IP02: A     #t_Safety_Pwr_On_GRP16;
      AN    #t_Suppress_Errors;
      AN    #t_Suppress_Errors_Isafe;
      AN    #s_Status.THO_Main_Pwr_GRP16;
      AN    #s_Status.No_Power_GRP16;
      AN    #s_Status.THO_Aux_Pwr_GRP16;
      A     #i_CFG_Motor_Prsnt_GRP16;
      =     #s_Motor_Grp.Motor_Group_16_in;
NETWORK
TITLE =JA: Safety Signal Handling
//Handle safety stop signals for every motor group
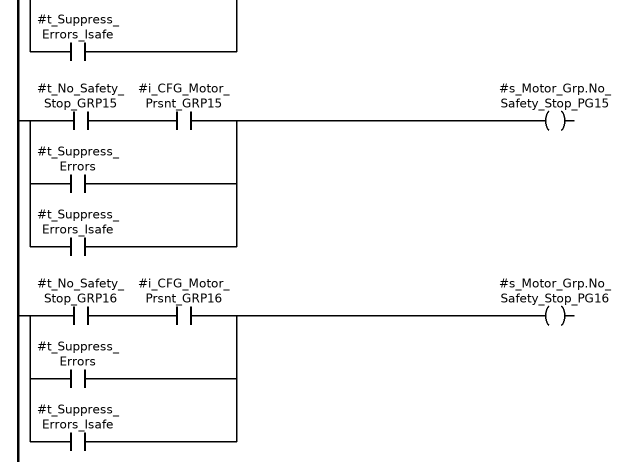
      NOP   0;
// No Safety stop MotorGroup 01
      A     #t_No_Safety_Stop_GRP01;
      A     #i_CFG_Motor_Prsnt_GRP01;
      O     #t_Suppress_Errors;
      O     #t_Suppress_Errors_Isafe;
      =     #s_Motor_Grp.No_Safety_Stop_PG01;

// No Safety stop MotorGroup 02
      A     #t_No_Safety_Stop_GRP02;
      A     #i_CFG_Motor_Prsnt_GRP02;
      O     #t_Suppress_Errors;
      O     #t_Suppress_Errors_Isafe;
      =     #s_Motor_Grp.No_Safety_Stop_PG02;

// No Safety stop MotorGroup 03
      A     #t_No_Safety_Stop_GRP03;
      A     #i_CFG_Motor_Prsnt_GRP03;
      O     #t_Suppress_Errors;
      O     #t_Suppress_Errors_Isafe;
      =     #s_Motor_Grp.No_Safety_Stop_PG03;

// No Safety stop MotorGroup 04
      A     #t_No_Safety_Stop_GRP04;
      A     #i_CFG_Motor_Prsnt_GRP04;
      O     #t_Suppress_Errors;
      O     #t_Suppress_Errors_Isafe;
      =     #s_Motor_Grp.No_Safety_Stop_PG04;

// No Safety stop MotorGroup 05
      A     #t_No_Safety_Stop_GRP05;
      A     #i_CFG_Motor_Prsnt_GRP05;
      O     #t_Suppress_Errors;
      O     #t_Suppress_Errors_Isafe;
      =     #s_Motor_Grp.No_Safety_Stop_PG05;

// No Safety stop MotorGroup 06
      A     #t_No_Safety_Stop_GRP06;
      A     #i_CFG_Motor_Prsnt_GRP06;
      O     #t_Suppress_Errors;
      O     #t_Suppress_Errors_Isafe;
      =     #s_Motor_Grp.No_Safety_Stop_PG06;

// No Safety stop MotorGroup 07
      A     #t_No_Safety_Stop_GRP07;
      A     #i_CFG_Motor_Prsnt_GRP07;
      O     #t_Suppress_Errors;
      O     #t_Suppress_Errors_Isafe;
      =     #s_Motor_Grp.No_Safety_Stop_PG07;

// No Safety stop MotorGroup 08
      A     #t_No_Safety_Stop_GRP08;
      A     #i_CFG_Motor_Prsnt_GRP08;
      O     #t_Suppress_Errors;
      O     #t_Suppress_Errors_Isafe;
      =     #s_Motor_Grp.No_Safety_Stop_PG08;

// No Safety stop MotorGroup 09
      A     #t_No_Safety_Stop_GRP09;
      A     #i_CFG_Motor_Prsnt_GRP09;
      O     #t_Suppress_Errors;
      O     #t_Suppress_Errors_Isafe;
      =     #s_Motor_Grp.No_Safety_Stop_PG09;

// No Safety stop MotorGroup 10
      A     #t_No_Safety_Stop_GRP10;
      A     #i_CFG_Motor_Prsnt_GRP10;
      O     #t_Suppress_Errors;
      O     #t_Suppress_Errors_Isafe;
      =     #s_Motor_Grp.No_Safety_Stop_PG10;

// No Safety stop MotorGroup 11
      A     #t_No_Safety_Stop_GRP11;
      A     #i_CFG_Motor_Prsnt_GRP11;
      O     #t_Suppress_Errors;
      O     #t_Suppress_Errors_Isafe;
      =     #s_Motor_Grp.No_Safety_Stop_PG11;

// No Safety stop MotorGroup 12
      A     #t_No_Safety_Stop_GRP12;
      A     #i_CFG_Motor_Prsnt_GRP12;
      O     #t_Suppress_Errors;
      O     #t_Suppress_Errors_Isafe;
      =     #s_Motor_Grp.No_Safety_Stop_PG12;

// No Safety stop MotorGroup 13
      A     #t_No_Safety_Stop_GRP13;
      A     #i_CFG_Motor_Prsnt_GRP13;
      O     #t_Suppress_Errors;
      O     #t_Suppress_Errors_Isafe;
      =     #s_Motor_Grp.No_Safety_Stop_PG13;

// No Safety stop MotorGroup 14
      A     #t_No_Safety_Stop_GRP14;
      A     #i_CFG_Motor_Prsnt_GRP14;
      O     #t_Suppress_Errors;
      O     #t_Suppress_Errors_Isafe;
      =     #s_Motor_Grp.No_Safety_Stop_PG14;

// No Safety stop MotorGroup 15
      A     #t_No_Safety_Stop_GRP15;
      A     #i_CFG_Motor_Prsnt_GRP15;
      O     #t_Suppress_Errors;
      O     #t_Suppress_Errors_Isafe;
      =     #s_Motor_Grp.No_Safety_Stop_PG15;

// No Safety stop MotorGroup 16
      A     #t_No_Safety_Stop_GRP16;
      A     #i_CFG_Motor_Prsnt_GRP16;
      O     #t_Suppress_Errors;
      O     #t_Suppress_Errors_Isafe;
      =     #s_Motor_Grp.No_Safety_Stop_PG16;

NETWORK
TITLE =KA: Copy motor group status to DB

      OPN   #i_DB_Motor_Slave;

      L     DBNO;
      T     #t_DB_NO;

      L     DBLG;
      T     #t_DB_Length;

// define t_ANY_data
      LAR1  P##t_ANY_DB_Motor_Slave; // input ANY POINTER

// Copy the the pointer type to the Temporary pointers
      L     W#16#1002; // ANY pointer type: 10 for S7, 02 for data type 'BYTE'
      T     LW [AR1,P#0.0]; // ANY pointer type

// Copy the repetition factor (= data lentgh) to the Temporary pointers
      L     #t_DB_Length; // Number of bytes to copy
      T     LW [AR1,P#2.0]; // ANY pointer repetition factor

// Copy the DB number to the Data temporary pointer
      L     #t_DB_NO; // ANY POINTER for data to write
      T     LW [AR1,P#4.0]; // ANY pointer DB number

// Copy the Area pointer to the Data Temporary pointer
      L     0;
      T     LD [AR1,P#6.0]; // ANY pointer Area pointer
      L     B#16#84; //Store 84H: DB Global data area in ANY
      T     LB [AR1,P#6.0];

      CALL "BLKMOV" (
           SRCBLK                   := #s_Motor_Grp,
           RET_VAL                  := #t_Ret_Val,
           DSTBLK                   := #t_ANY_DB_Motor_Slave);

NETWORK
TITLE =LA: Handle commands
//Set the controlled stop and direct stop output signals.
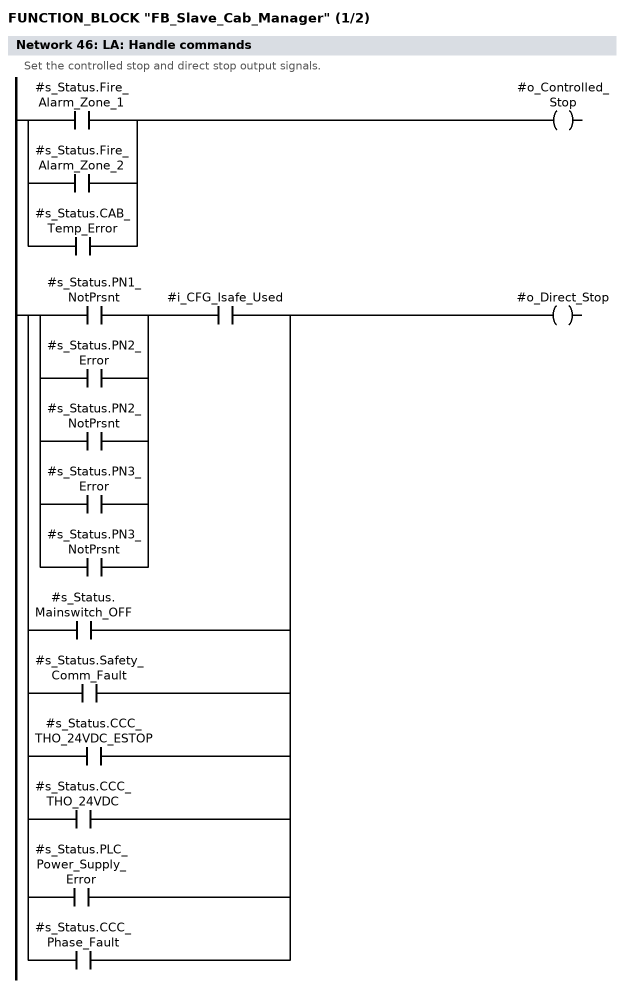
      O     #s_Status.Fire_Alarm_Zone_1;
      O     #s_Status.Fire_Alarm_Zone_2;
      O     #s_Status.CAB_Temp_Error;
      =     #o_Controlled_Stop;

      A(    ;
      O     #s_Status.PN1_NotPrsnt;
      O     #s_Status.PN2_Error;
      O     #s_Status.PN2_NotPrsnt;
      O     #s_Status.PN3_Error;
      O     #s_Status.PN3_NotPrsnt;
      )     ;
      A     #i_CFG_Isafe_Used;
      O     #s_Status.Mainswitch_OFF;
      O     #s_Status.Safety_Comm_Fault;
      O     #s_Status.CCC_THO_24VDC_ESTOP;
      O     #s_Status.CCC_THO_24VDC;
      O     #s_Status.PLC_Power_Supply_Error;
// Option to stop is Phase fault is detected.
      O     #s_Status.CCC_Phase_Fault;
      =     #o_Direct_Stop;
NETWORK
TITLE =MA: Write output signals
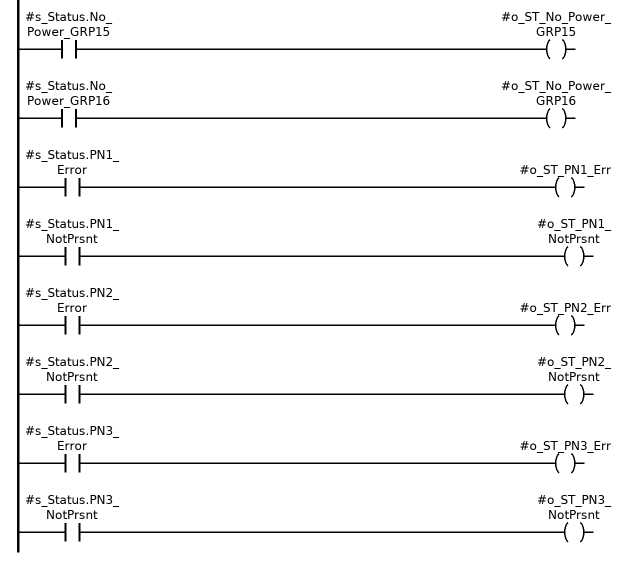

      A     #s_Status.Mainswitch_OFF;
      =     #o_ST_Mainswitch_OFF;

      A     #s_Status.Safety_Comm_Fault;
      =     #o_ST_Safety_Comm_Fault;

      A     #s_Status.CCC_THO_24VDC;
      =     #o_ST_CCC_THO_1_24VDC;

      A     #s_Status.PLC_Power_Supply_Error;
      =     #o_ST_CCC_THO_2_24VDC;

      A     #s_Status.CCC_THO_24VDC_ESTOP;
      =     #o_ST_CCC_THO_24VDC_ESTOP;

      A     #s_Status.CCC_THO_Phase;
      =     #o_ST_CCC_THO_Phase;

      A     #s_Status.CCC_Phase_Fault;
      =     #o_ST_CCC_Phase_Fault;

      A     #s_Status.Fire_Alarm_Zone_1;
      =     #o_ST_Fire_Alarm_Zone_1;

      A     #s_Status.Fire_Alarm_Zone_2;
      =     #o_ST_Fire_Alarm_Zone_2;

      A     #s_Status.ETH_Switch_Fault;
      =     #o_ST_ETH_Switch_Fault;

      A     #s_Status.CAB_Temp_High;
      =     #o_ST_CAB_Temp_High;

      A     #s_Status.CAB_Temp_Error;
      =     #o_ST_CAB_Temp_Error;

      A     #s_Status.UPS_THO;
      =     #o_ST_UPS_THO;

      A     #s_Status.THO_Main_Pwr_GRP01;
      =     #o_ST_THO_Main_Pwr_GRP01;

      A     #s_Status.THO_Main_Pwr_GRP02;
      =     #o_ST_THO_Main_Pwr_GRP02;

      A     #s_Status.THO_Main_Pwr_GRP03;
      =     #o_ST_THO_Main_Pwr_GRP03;

      A     #s_Status.THO_Main_Pwr_GRP04;
      =     #o_ST_THO_Main_Pwr_GRP04;

      A     #s_Status.THO_Main_Pwr_GRP05;
      =     #o_ST_THO_Main_Pwr_GRP05;

      A     #s_Status.THO_Main_Pwr_GRP06;
      =     #o_ST_THO_Main_Pwr_GRP06;

      A     #s_Status.THO_Main_Pwr_GRP07;
      =     #o_ST_THO_Main_Pwr_GRP07;

      A     #s_Status.THO_Main_Pwr_GRP08;
      =     #o_ST_THO_Main_Pwr_GRP08;

      A     #s_Status.THO_Main_Pwr_GRP09;
      =     #o_ST_THO_Main_Pwr_GRP09;

      A     #s_Status.THO_Main_Pwr_GRP10;
      =     #o_ST_THO_Main_Pwr_GRP10;

      A     #s_Status.THO_Main_Pwr_GRP11;
      =     #o_ST_THO_Main_Pwr_GRP11;

      A     #s_Status.THO_Main_Pwr_GRP12;
      =     #o_ST_THO_Main_Pwr_GRP12;

      A     #s_Status.THO_Main_Pwr_GRP13;
      =     #o_ST_THO_Main_Pwr_GRP13;

      A     #s_Status.THO_Main_Pwr_GRP14;
      =     #o_ST_THO_Main_Pwr_GRP14;

      A     #s_Status.THO_Main_Pwr_GRP15;
      =     #o_ST_THO_Main_Pwr_GRP15;

      A     #s_Status.THO_Main_Pwr_GRP16;
      =     #o_ST_THO_Main_Pwr_GRP16;

      A     #s_Status.THO_Aux_Pwr_GRP01;
      =     #o_ST_THO_Aux_Pwr_GRP01;

      A     #s_Status.THO_Aux_Pwr_GRP02;
      =     #o_ST_THO_Aux_Pwr_GRP02;

      A     #s_Status.THO_Aux_Pwr_GRP03;
      =     #o_ST_THO_Aux_Pwr_GRP03;

      A     #s_Status.THO_Aux_Pwr_GRP04;
      =     #o_ST_THO_Aux_Pwr_GRP04;

      A     #s_Status.THO_Aux_Pwr_GRP05;
      =     #o_ST_THO_Aux_Pwr_GRP05;

      A     #s_Status.THO_Aux_Pwr_GRP06;
      =     #o_ST_THO_Aux_Pwr_GRP06;

      A     #s_Status.THO_Aux_Pwr_GRP07;
      =     #o_ST_THO_Aux_Pwr_GRP07;

      A     #s_Status.THO_Aux_Pwr_GRP08;
      =     #o_ST_THO_Aux_Pwr_GRP08;

      A     #s_Status.THO_Aux_Pwr_GRP09;
      =     #o_ST_THO_Aux_Pwr_GRP09;

      A     #s_Status.THO_Aux_Pwr_GRP10;
      =     #o_ST_THO_Aux_Pwr_GRP10;

      A     #s_Status.THO_Aux_Pwr_GRP11;
      =     #o_ST_THO_Aux_Pwr_GRP11;

      A     #s_Status.THO_Aux_Pwr_GRP12;
      =     #o_ST_THO_Aux_Pwr_GRP12;

      A     #s_Status.THO_Aux_Pwr_GRP13;
      =     #o_ST_THO_Aux_Pwr_GRP13;

      A     #s_Status.THO_Aux_Pwr_GRP14;
      =     #o_ST_THO_Aux_Pwr_GRP14;

      A     #s_Status.THO_Aux_Pwr_GRP15;
      =     #o_ST_THO_Aux_Pwr_GRP15;

      A     #s_Status.THO_Aux_Pwr_GRP16;
      =     #o_ST_THO_Aux_Pwr_GRP16;

      A     #s_Status.No_Power_GRP01;
      =     #o_ST_No_Power_GRP01;

      A     #s_Status.No_Power_GRP02;
      =     #o_ST_No_Power_GRP02;

      A     #s_Status.No_Power_GRP03;
      =     #o_ST_No_Power_GRP03;

      A     #s_Status.No_Power_GRP04;
      =     #o_ST_No_Power_GRP04;

      A     #s_Status.No_Power_GRP05;
      =     #o_ST_No_Power_GRP05;

      A     #s_Status.No_Power_GRP06;
      =     #o_ST_No_Power_GRP06;

      A     #s_Status.No_Power_GRP07;
      =     #o_ST_No_Power_GRP07;

      A     #s_Status.No_Power_GRP08;
      =     #o_ST_No_Power_GRP08;

      A     #s_Status.No_Power_GRP09;
      =     #o_ST_No_Power_GRP09;

      A     #s_Status.No_Power_GRP10;
      =     #o_ST_No_Power_GRP10;

      A     #s_Status.No_Power_GRP11;
      =     #o_ST_No_Power_GRP11;

      A     #s_Status.No_Power_GRP12;
      =     #o_ST_No_Power_GRP12;

      A     #s_Status.No_Power_GRP13;
      =     #o_ST_No_Power_GRP13;

      A     #s_Status.No_Power_GRP14;
      =     #o_ST_No_Power_GRP14;

      A     #s_Status.No_Power_GRP15;
      =     #o_ST_No_Power_GRP15;

      A     #s_Status.No_Power_GRP16;
      =     #o_ST_No_Power_GRP16;

      A     #s_Status.PN1_Error;
      =     #o_ST_PN1_Err;

      A     #s_Status.PN1_NotPrsnt;
      =     #o_ST_PN1_NotPrsnt;

      A     #s_Status.PN2_Error;
      =     #o_ST_PN2_Err;

      A     #s_Status.PN2_NotPrsnt;
      =     #o_ST_PN2_NotPrsnt;

      A     #s_Status.PN3_Error;
      =     #o_ST_PN3_Err;

      A     #s_Status.PN3_NotPrsnt;
      =     #o_ST_PN3_NotPrsnt;

END_FUNCTION_BLOCK

